TYPE E_SlaveArmState :
(
	SlaveArmState_Error := 1,
	SlaveArmState_SelfCheck :=2,
	SlaveArmState_Init :=3,
	SlaveArmState_Standby :=4,
	SlaveArmState_InstallPanel:=5,
	SlaveArmState_PanelReady :=6,
	SlaveArmState_InstallInstru :=7,
	SlaveArmState_InstruReady :=8,
	SlaveArmState_MasterSlave :=9,
	SlaveArmState_InstallScope :=10,
	SlaveArmState_ScopeReady :=11,
	SlaveArmState_EndoScope :=12,
	SlaveArmState_Cart := 13
);
END_TYPE

(* stored: Version 1.1.0.1, ProductVersion 3.1.4024.12
   DUT E_SlaveArmState: Id {1989848d-a357-4300-a3bc-ded8b39d8e17} *)
